ABB RAPID module: Module1.mod

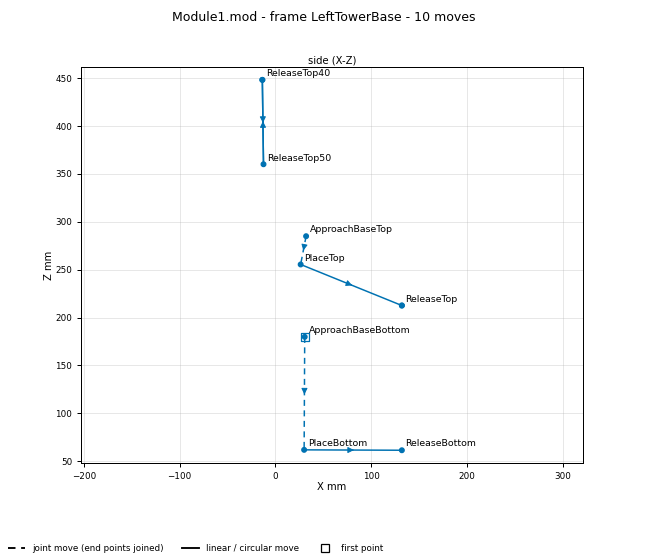
[picture p0: tool path of Module1.mod in frame LeftTowerBase, 10 of 25 moves have a stored position in this frame; points joined in program order, loops and branches not executed]
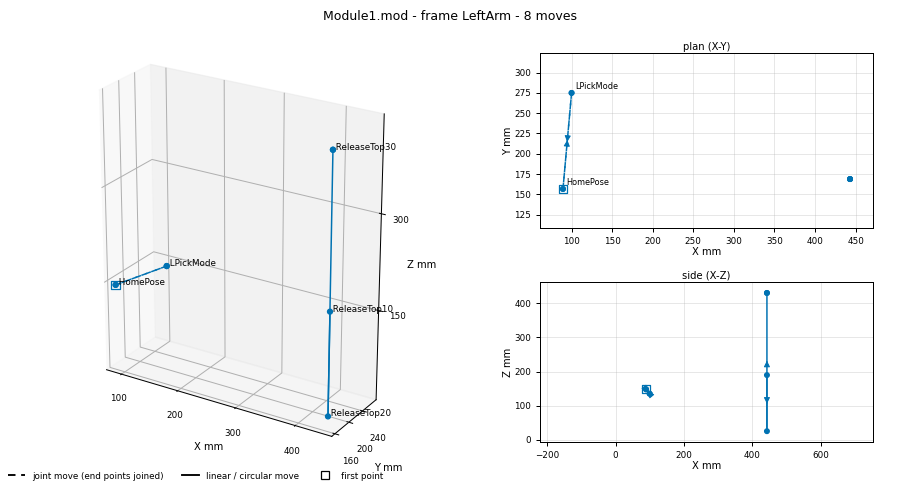
[picture p1: tool path of Module1.mod in frame LeftArm, 8 of 25 moves have a stored position in this frame; points joined in program order, loops and branches not executed]
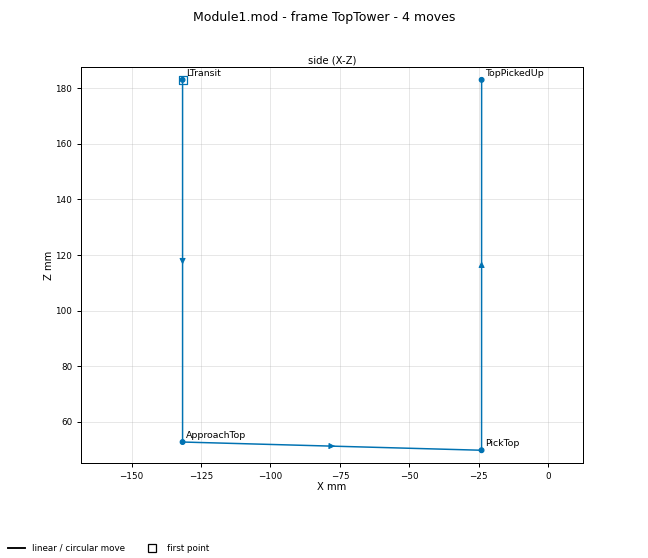
[picture p2: tool path of Module1.mod in frame TopTower, 4 of 25 moves have a stored position in this frame; points joined in program order, loops and branches not executed]
MODULE Module1
    CONST robtarget HomePose:=[[89.387946423,156.622117957,147.913470217],[0.066010726,0.842420918,-0.111214912,0.523068661],[0,0,-1,4],[101.964427132,9E+09,9E+09,9E+09,9E+09,9E+09]];
    CONST robtarget LPickMode:=[[100,275,135],[0.489762134,0.473830049,0.544432409,0.489092516],[0,0,0,4],[106.3570107,9E+09,9E+09,9E+09,9E+09,9E+09]];
    CONST robtarget ApproachBottom:=[[-123.000341943,0.00869998,49.700265433],[0.500019373,0.500017356,0.499980624,0.499982645],[0,0,-1,4],[101.964431609,9E+09,9E+09,9E+09,9E+09,9E+09]];
    CONST robtarget PickBottom:=[[-32.000174,0.0028828,49.699574469],[0.500019373,0.500017356,0.499980624,0.499982645],[-1,0,-1,4],[101.964431609,9E+09,9E+09,9E+09,9E+09,9E+09]];
    CONST robtarget BottomPickedUp:=[[-32.000042144,-0.000088177,183.047951174],[0.5000156,0.500018782,0.499980217,0.499985399],[0,0,-1,4],[101.964431609,9E+09,9E+09,9E+09,9E+09,9E+09]];
    CONST robtarget ApproachBaseBottom:=[[30.55,0.33,179.86],[0.497467,0.501702,-0.503099,-0.497708],[-1,1,-2,4],[101.938,9E+09,9E+09,9E+09,9E+09,9E+09]];
    CONST robtarget PlaceBottom:=[[29.94,0.02,61.87],[0.499995,0.499995,-0.499999,-0.500011],[-1,1,-2,4],[101.931,9E+09,9E+09,9E+09,9E+09,9E+09]];
    CONST robtarget ReleaseBottom:=[[132,0,61.45],[0.5,0.5,-0.5,-0.5],[-1,1,-2,4],[101.964435132,9E+09,9E+09,9E+09,9E+09,9E+09]];
    CONST robtarget LTransit:=[[-131.628352317,0.395873729,183.048301566],[0.500280603,0.500280878,0.499719692,0.499718512],[-1,1,-2,4],[101.964432039,9E+09,9E+09,9E+09,9E+09,9E+09]];
    CONST robtarget ApproachTop:=[[-131.629543032,0.394757125,52.700301569],[0.500280603,0.500280878,0.499719692,0.499718512],[0,0,-1,4],[101.964432039,9E+09,9E+09,9E+09,9E+09,9E+09]];
    CONST robtarget PickTop:=[[-24.02,0.01,49.74],[0.500276,0.500285,0.499723,0.499716],[-1,0,-1,4],[101.963,9E+09,9E+09,9E+09,9E+09,9E+09]];
    CONST robtarget TopPickedUp:=[[-23.999717886,0.009976627,183.048145368],[0.500280603,0.500280878,0.499719692,0.499718512],[-1,0,-1,4],[101.964432039,9E+09,9E+09,9E+09,9E+09,9E+09]];
    CONST robtarget ApproachBaseTop:=[[32,0,285],[0.5,0.5,-0.5,-0.5],[-1,0,-2,4],[101.964431609,9E+09,9E+09,9E+09,9E+09,9E+09]];
    CONST robtarget PlaceTop:=[[26.30,3.05,255.47],[0.500002,0.49999,-0.500002,-0.500006],[-1,1,-2,4],[101.961,9E+09,9E+09,9E+09,9E+09,9E+09]];
    CONST robtarget ReleaseTop:=[[132,0,212.6],[0.5,0.5,-0.5,-0.5],[-1,1,-2,4],[101.964430108,9E+09,9E+09,9E+09,9E+09,9E+09]];
    VAR syncident sync1;
    PERS tasks tasklist1{2}:=[["T_ROB_L"],["T_ROB_R"]];
    VAR syncident sync2;
    VAR syncident sync3;
    CONST robtarget ReleaseTop10:=[[443.09,168.87,189.52],[1.84955E-05,0.711078,-0.703113,1.6546E-05],[-1,2,-1,4],[120.086,9E+09,9E+09,9E+09,9E+09,9E+09]];
    CONST robtarget ReleaseTop20:=[[443.05,168.79,25.36],[0.000552156,0.710906,-0.703287,0.000279454],[-1,2,-1,4],[120.096,9E+09,9E+09,9E+09,9E+09,9E+09]];
    CONST robtarget ReleaseTop30:=[[443.07,168.82,429.89],[0.000113649,0.710991,-0.703201,1.61698E-05],[-1,1,-2,4],[149.06,9E+09,9E+09,9E+09,9E+09,9E+09]];
    CONST robtarget ReleaseTop40:=[[-13.70,0.74,448.28],[0.000915826,0.687079,0.726582,-0.000107677],[-1,1,-1,4],[171.886,9E+09,9E+09,9E+09,9E+09,9E+09]];
    CONST robtarget ReleaseTop50:=[[-12.49,-1.11,360.13],[0.00827057,-0.689573,-0.724016,-0.0148913],[-1,1,-1,4],[172.058,9E+09,9E+09,9E+09,9E+09,9E+09]];
    VAR syncident sync4;
    PROC Path_10()
        ConfJ\Off;
        ConfL\Off;
        MoveJ HomePose,v100,fine,Servo\WObj:=LeftArm;
        MoveJ LPickMode,v100,fine,Servo\WObj:=LeftArm;
        g_MoveTo 4;
        MoveJ ApproachBottom,v100,fine,Servo\WObj:=BottomTower;
        MoveL PickBottom,v100,fine,Servo\WObj:=BottomTower;
        g_GripIn;
        WaitTime 1;
        MoveL BottomPickedUp,v100,fine,Servo\WObj:=BottomTower;
        MoveL ApproachBaseBottom,v100,fine,Servo\WObj:=LeftTowerBase;
        MoveJ PlaceBottom,v100,fine,Servo\WObj:=LeftTowerBase;
        WaitSyncTask\InPos, sync1, tasklist1;
        g_MoveTo 4;
        WaitTime 1;
        MoveL ReleaseBottom,v100,fine,Servo\WObj:=LeftTowerBase;
        MoveL LTransit,v100,fine,Servo\WObj:=TopTower;
        MoveL ApproachTop,v100,fine,Servo\WObj:=TopTower;
        MoveL PickTop,v100,fine,Servo\WObj:=TopTower;
        g_GripIn;
        WaitTime 1;
        MoveL TopPickedUp,v100,fine,Servo\WObj:=TopTower;
        MoveJ ApproachBaseTop,v100,fine,Servo\WObj:=LeftTowerBase;
        MoveJ PlaceTop,v100,fine,Servo\WObj:=LeftTowerBase;
        WaitSyncTask\InPos, sync2, tasklist1;
        g_MoveTo 4;
        WaitTime 1;
        MoveL ReleaseTop,v100,fine,Servo\WObj:=LeftTowerBase;
        MoveJ ReleaseTop10, v100, fine, Servo\WObj:=LeftArm;
        g_GripOut;
        WaitTime 1;
        MoveL ReleaseTop20, v100, fine, Servo\WObj:=LeftArm;
        g_GripIn;
        WaitTime 1;
        WaitSyncTask\InPos, sync3, tasklist1;
        MoveL ReleaseTop30, v100, fine, Servo\WObj:=LeftArm;
        WaitSyncTask\InPos, sync4, tasklist1;
        MoveL ReleaseTop40, v100, fine, Servo\WObj:=LeftTowerBase;
        MoveL ReleaseTop50, v100, fine, Servo\WObj:=LeftTowerBase;
        g_GripOut;
        WaitTime 1;
        MoveL ReleaseTop40, v100, fine, Servo\WObj:=LeftTowerBase;
        MoveL ReleaseTop30, v100, fine, Servo\WObj:=LeftArm;
        MoveL ReleaseTop,v100,fine,Servo\WObj:=LeftTowerBase;
        MoveJ LPickMode,v100,fine,Servo\WObj:=LeftArm;
        MoveJ HomePose,v100,fine,Servo\WObj:=LeftArm;
    ENDPROC
ENDMODULE
